// TIA Portal V20 export
DATA_BLOCK "LBP_MFuncDecListConfig"   // DB75
TITLE = M decoding acc. to list / Décodage M selon liste
{ S7_Optimized_Access := 'FALSE' }
AUTHOR : SINUMERIK
FAMILY : SINUMERIK_ONE
VERSION : 6.24
// Interface between user program and NCK, contains the configuration for the M functions to be decoded / Interface entre programme utilisateur et NCK contient la configuration des fonctions M à décoder.
// stored: AutoNumber false
   VAR RETAIN
      MSigGrp : Array[1..16] of Struct
         MExtAdr : Int;
         MFirstAdr : DInt;
         MLastAdr : DInt;
      END_STRUCT;
   END_VAR
BEGIN
   MSigGrp[1..16].MFirstAdr := DINT#0;
   MSigGrp[1..16].MLastAdr := DINT#0;
END_DATA_BLOCK
